// TwinCAT 3 PLC project PLC1
// ProgramVersion: 3.1.4024.0
// libraries:
//   Tc2_Standard, * (Beckhoff Automation GmbH)
//   Tc2_System, * (Beckhoff Automation GmbH)
//   Tc3_Module, * (Beckhoff Automation GmbH)
//   VisuDialogs, * (System)
//   VisuSymbols,3.5.10.0,System
// project tree:
//   / GlobalTextList.TcGTLO, PlcTask.TcTTO, Visualization Manager.TcVMO (not stored)
//   GVLs/ Cell.TcGVL, SEQ.TcGVL, VAL.TcGVL, Variables.TcGVL
//   POUs/ MAIN.TcPOU, POU.TcPOU, POU_1.TcPOU, FBAdd.TcPOU, Func.TcPOU, POU_3.TcPOU, SequencyControl.TcPOU, Simulation.TcPOU, ValveControl.TcPOU, Water_Tank.TcPOU
//   VISUs/ Header.TcVIS, MainScreen.TcVIS, Nav.TcVIS, Visualization.TcVIS, Visualization_1.TcVIS
// real-time tasks:
//   TASK PlcTask: cycle T#10ms, priority 20, ADS port 350
//   TASK VISU_TASK: cycle T#200000us, priority 30, ADS port 351

CONFIGURATION PLC1
    RESOURCE PLC ON TwinCAT3
        TASK PlcTask(INTERVAL := T#10ms, PRIORITY := 20);
        PROGRAM MAIN WITH PlcTask : MAIN;
    END_RESOURCE
END_CONFIGURATION

// ---- GVLs/Cell.TcGVL
{attribute 'qualified_only'}
VAR_GLOBAL
	bPalmButton:BOOL;
	bHousingPresent:BOOL;
	
END_VAR

// ---- GVLs/SEQ.TcGVL
{attribute 'qualified_only'}
VAR_GLOBAL
	iStepN:WORD;
	iSeqStepN: INT;
	sSeqStepDescription: STRING;
	bSeqStep_TaskDone: ARRAY[0..30] OF BOOL;
	fbSeqStepN_TaskDone_DelayTmr:ARRAY[0..30] OF TON;
	bSeqStepN_TaskDone_DelayDone:ARRAY[0..30] OF BOOL;

END_VAR

// ---- GVLs/VAL.TcGVL
{attribute 'qualified_only'}
VAR_GLOBAL
	bValve_A_WorkCmd:BOOL;
	bValve_A_HomeCmd:BOOL;
	bValve_A_AtWorkSensor:BOOL;
	bValve_A_AtHomeSensor:BOOL;
	
    bValve_B_WorkCmd:BOOL;
	bValve_B_HomeCmd:BOOL;
	bValve_B_AtWorkSensor:BOOL;
	bValve_B_AtHomeSensor:BOOL;
	
	bValve_C_WorkCmd:BOOL;
	bValve_C_HomeCmd:BOOL;
	bValve_C_AtWorkSensor:BOOL;
	bValve_C_AtHomeSensor:BOOL;
	
	bValve_D_WorkCmd:BOOL;
	bValve_D_HomeCmd:BOOL;
	bValve_D_AtWorkSensor:BOOL;
	bValve_D_AtHomeSensor:BOOL;
	
	bAllValves_At_Home:BOOL;
	
END_VAR

// ---- GVLs/Variables.TcGVL
{attribute 'qualified_only'}
VAR_GLOBAL
	stop:BOOL;
	start:BOOL;
	motor1:BOOL;
	motor2:BOOL;
	motor3:BOOL;
	LED:BOOL;
	Button:BOOL;
	Temp:BOOL;
END_VAR

// ---- POUs/MAIN.TcPOU
PROGRAM MAIN
VAR
END_VAR

SEQ.iStepN:=30;
Simulation();
POU();
Water_Tank();
POU_1();
POU_3();
SequencyControl();
ValveControl();

END_PROGRAM

// ---- POUs/Simulation.TcPOU
PROGRAM Simulation
VAR
END_VAR

VAL.bValve_A_AtHomeSensor:=VAL.bValve_A_HomeCmd;
VAL.bValve_A_AtWorkSensor:=VAL.bValve_A_WorkCmd;

VAL.bValve_B_AtHomeSensor:=VAL.bValve_B_HomeCmd;
VAL.bValve_B_AtWorkSensor:=VAL.bValve_B_WorkCmd;

VAL.bValve_C_AtHomeSensor:=VAL.bValve_C_HomeCmd;
VAL.bValve_C_AtWorkSensor:=VAL.bValve_C_WorkCmd;

VAL.bValve_D_AtHomeSensor:=VAL.bValve_D_HomeCmd;
VAL.bValve_D_AtWorkSensor:=VAL.bValve_D_WorkCmd;

END_PROGRAM

// ---- POUs/POU.TcPOU
PROGRAM POU
VAR
	T1: TON;
	TON_0:TON;
    Cycle: BOOL;
END_VAR
VAR // added by the converter: edge detectors and wires of the graphical bodies
    _w1 : BOOL;
END_VAR

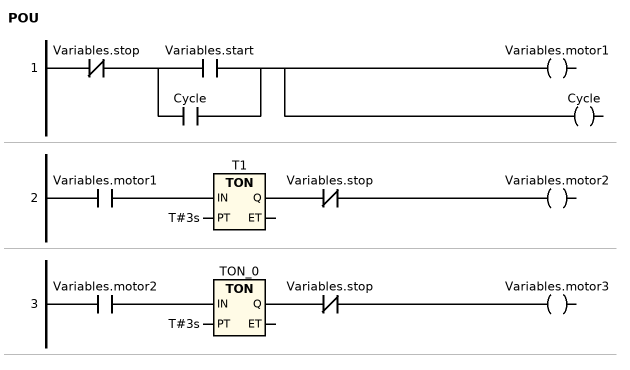
// NETWORK 1
_w1 := NOT Variables.stop AND (Variables.start OR Cycle);
Variables.motor1 := _w1;
Cycle := _w1;

// NETWORK 2
T1(IN := Variables.motor1, PT := T#3s); // TON
Variables.motor2 := T1.Q AND NOT Variables.stop;

// NETWORK 3
TON_0(IN := Variables.motor2, PT := T#3s); // TON
Variables.motor3 := TON_0.Q AND NOT Variables.stop;

END_PROGRAM

// ---- POUs/Water_Tank.TcPOU
PROGRAM Water_Tank
VAR
	start:BOOL;
	stop:BOOL;
	high:BOOL;
	low:BOOL;
	motor:BOOL;
	temp:BOOL;
	mix:BOOL;
	release:BOOL;
	
	TON_0: TON;
	TOF_0: TOF;
	TON_1: TON;
	MixFor10S: TOF;
	Delay2S: TON;
END_VAR

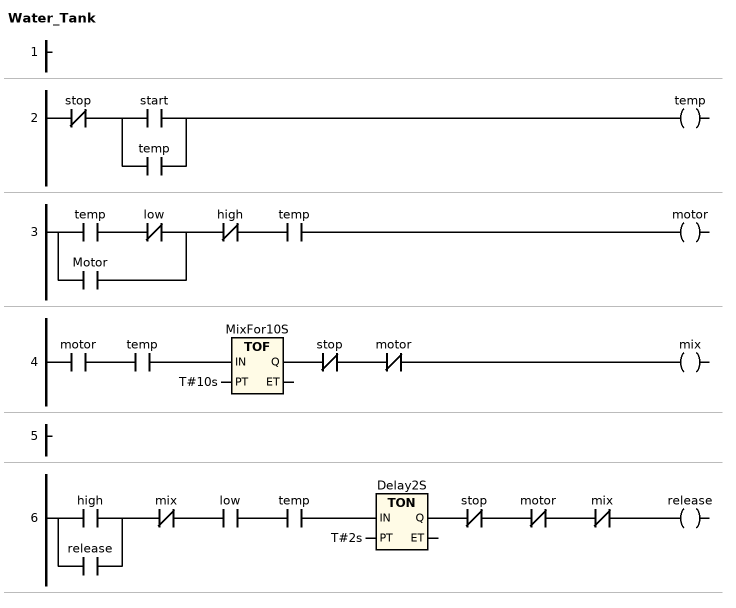
// NETWORK 1

// NETWORK 2
temp := NOT stop AND (start OR temp);

// NETWORK 3
motor := (temp AND NOT low OR Motor) AND NOT high AND temp;

// NETWORK 4
MixFor10S(IN := motor AND temp, PT := T#10s); // TOF
mix := MixFor10S.Q AND NOT stop AND NOT motor;

// NETWORK 5

// NETWORK 6
Delay2S(IN := (high OR release) AND NOT mix AND low AND temp, PT := T#2s); // TON
release := Delay2S.Q AND NOT stop AND NOT motor AND NOT mix;

END_PROGRAM

// ---- POUs/POU_1.TcPOU
PROGRAM POU_1
VAR
	x:BOOL;
	y:BOOL;
     rr:BOOL;
	 ss:bool;
	counter: CTU;
	coun:WORD;
END_VAR

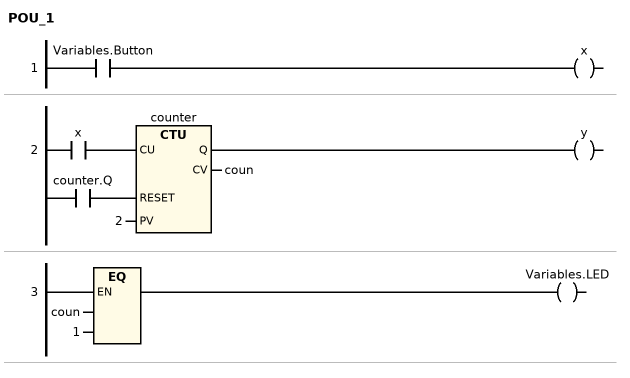
// NETWORK 1
x := Variables.Button;

// NETWORK 2
counter(CU := x, RESET := counter.Q, PV := 2, CV => coun); // CTU
y := counter.Q;

// NETWORK 3
Variables.LED := coun = 1;

END_PROGRAM

// ---- POUs/POU_3.TcPOU
PROGRAM POU_3
VAR
	count:WORD;
	prePushed:BOOL;
	pre: INT;
	fbCal:FBAdd;
	result:WORD;
	x:WORD;
	y:WORD;
	z:word;
END_VAR


IF Variables.Button THEN 
	IF NOT prePushed THEN
		count:=count+1;
		prePushed:=TRUE;
		Variables.LED:=NOT Variables.LED;
	END_IF
ELSE
	prePushed:=FALSE;	
END_IF
	
fbCal(a:=5,b:=3,c=>result);


x:=4;
y:=7;
//count:=Func(1,4);
z:=Func(x,y);

ACTION ACT:

END_ACTION

METHOD PUBLIC METH : BOOL
VAR_INPUT
END_VAR
END_METHOD

METHOD PUBLIC METH_1 : BOOL
VAR_INPUT
END_VAR
END_METHOD

END_PROGRAM

// ---- POUs/FBAdd.TcPOU
FUNCTION_BLOCK FINAL FBAdd
VAR_INPUT
	a:WORD;
	b:WORD;
END_VAR
VAR_OUTPUT
	c:word;
END_VAR
VAR
END_VAR

c:=a+b;
c:=a*b;

ACTION ACT:

END_ACTION

METHOD PUBLIC METH : BOOL
VAR_INPUT
END_VAR
END_METHOD

METHOD PRIVATE METH_1 : BOOL
VAR_INPUT
END_VAR
END_METHOD

PROPERTY PUBLIC Prop : INT
GET
END_GET
SET
END_SET
END_PROPERTY

END_FUNCTION_BLOCK

// ---- POUs/Func.TcPOU
FUNCTION Func : WORD
VAR_INPUT
	a:WORD;
	b:WORD;
END_VAR
VAR
	c:WORD;
END_VAR

c:=a+b;
Func:=c;
RETURN;

END_FUNCTION

// ---- POUs/SequencyControl.TcPOU
PROGRAM SequencyControl
VAR
	index:WORD;
END_VAR

CASE SEQ.iSeqStepN OF 
	 0:    //INIT
		 SEQ.sSeqStepDescription:='Init';
		 SEQ.bSeqStep_TaskDone[0]:=VAL.bAllValves_At_Home AND Cell.bHousingPresent AND Cell.bPalmButton;  //trigger the sequency
		 IF SEQ.bSeqStepN_TaskDone_DelayDone[0] THEN
			 FOR index:=1 TO SEQ.iStepN DO
				 SEQ.bSeqStep_TaskDone[index]:=FALSE;
			 END_FOR
			 seq.iSeqStepN:=5;
		 END_IF
	5:
		 SEQ.sSeqStepDescription:='Loading parts to hoursing';
		 SEQ.bSeqStep_TaskDone[5]:=VAL.bValve_A_AtWorkSensor;
		 IF SEQ.bSeqStepN_TaskDone_DelayDone[5] THEN
			 FOR index:=6 TO SEQ.iStepN DO
				 SEQ.bSeqStep_TaskDone[index]:=FALSE;
			 END_FOR
			 seq.iSeqStepN:=10;
		 END_IF
	10:
		 SEQ.sSeqStepDescription:='Clamp house';
		 SEQ.bSeqStep_TaskDone[10]:=VAL.bValve_A_AtWorkSensor AND VAl.bValve_B_AtWorkSensor;
		 IF SEQ.bSeqStepN_TaskDone_DelayDone[10] THEN
			 FOR index:=11 TO SEQ.iStepN DO
				 SEQ.bSeqStep_TaskDone[index]:=FALSE;
			 END_FOR
			 seq.iSeqStepN:=15;
		 END_IF
	15:
  	     SEQ.sSeqStepDescription:='Press/crimp the housing';
		 SEQ.bSeqStep_TaskDone[15]:=VAL.bValve_B_AtWorkSensor AND VAL.bValve_C_AtWorkSensor AND VAL.bValve_A_AtHomeSensor;
		 IF SEQ.bSeqStepN_TaskDone_DelayDone[15] THEN
			 FOR index:=0 TO SEQ.iStepN DO
				 SEQ.bSeqStep_TaskDone[index]:=FALSE;
			 END_FOR
			 seq.iSeqStepN:=20;
		 END_IF
	20:
  	     SEQ.sSeqStepDescription:='Open clamp';
		 SEQ.bSeqStep_TaskDone[20]:=VAl.bValve_B_AtHomeSensor;
		 IF SEQ.bSeqStepN_TaskDone_DelayDone[20] THEN
			 FOR index:=21 TO SEQ.iStepN DO
				 SEQ.bSeqStep_TaskDone[index]:=FALSE;
			 END_FOR
			 seq.iSeqStepN:=25;
		 END_IF
	25:  //work on cyl D
		 SEQ.sSeqStepDescription:='Heat houring for 10s';
		 SEQ.bSeqStep_TaskDone[25]:=VAL.bValve_D_AtWorkSensor AND VAL.bValve_C_AtWorkSensor;
		 IF SEQ.bSeqStepN_TaskDone_DelayDone[25] THEN
			 FOR index:=26 TO SEQ.iStepN DO
				 SEQ.bSeqStep_TaskDone[index]:=FALSE;
			 END_FOR
			 seq.iSeqStepN:=30;
		 END_IF
	30:  //home, home cyn C and Cyn B
		 SEQ.sSeqStepDescription:='Stop heat, open clamp';
		 SEQ.bSeqStep_TaskDone[30]:=VAL.bValve_C_AtHomeSensor AND VAL.bValve_D_AtHomeSensor;
		 IF SEQ.bSeqStepN_TaskDone_DelayDone[30] THEN
//			 FOR index:=26 TO SEQ.iStepN DO
//				 SEQ.bSeqStep_TaskDone[index]:=FALSE;
//			 END_FOR
			 seq.iSeqStepN:=0;
		 END_IF
END_CASE
SequencyCondition();

METHOD PUBLIC SequencyCondition : BOOL
VAR_INPUT
END_VAR
SEQ.fbSeqStepN_TaskDone_DelayTmr[0](IN:= SEQ.bSeqStep_TaskDone[0], PT:=T#2S , Q=>SEQ.bSeqStepN_TaskDone_DelayDone[0] );
SEQ.fbSeqStepN_TaskDone_DelayTmr[5](IN:= SEQ.bSeqStep_TaskDone[5], PT:=T#2S , Q=>SEQ.bSeqStepN_TaskDone_DelayDone[5] );
SEQ.fbSeqStepN_TaskDone_DelayTmr[10](IN:= SEQ.bSeqStep_TaskDone[10], PT:=T#2S , Q=>SEQ.bSeqStepN_TaskDone_DelayDone[10] );
SEQ.fbSeqStepN_TaskDone_DelayTmr[15](IN:= SEQ.bSeqStep_TaskDone[15], PT:=T#2S , Q=>SEQ.bSeqStepN_TaskDone_DelayDone[15] );
SEQ.fbSeqStepN_TaskDone_DelayTmr[20](IN:= SEQ.bSeqStep_TaskDone[20], PT:=T#2S , Q=>SEQ.bSeqStepN_TaskDone_DelayDone[20] );
SEQ.fbSeqStepN_TaskDone_DelayTmr[25](IN:= SEQ.bSeqStep_TaskDone[25], PT:=T#10S , Q=>SEQ.bSeqStepN_TaskDone_DelayDone[25] );
SEQ.fbSeqStepN_TaskDone_DelayTmr[30](IN:= SEQ.bSeqStep_TaskDone[30], PT:=T#2S , Q=>SEQ.bSeqStepN_TaskDone_DelayDone[30] );
END_METHOD

END_PROGRAM

// ---- POUs/ValveControl.TcPOU
PROGRAM ValveControl
VAR
END_VAR

IF (SEQ.iSeqStepN=0 OR SEQ.iSeqStepN=30) THEN
	VAL.bValve_A_HomeCmd:=TRUE;
	VAL.bValve_A_WorkCmd:=FALSE;
	VAL.bValve_B_HomeCmd:=TRUE;
	VAL.bValve_B_WorkCmd:=FALSE;
	VAL.bValve_C_HomeCmd:=TRUE;
	VAL.bValve_C_WorkCmd:=FALSE;
	VAL.bValve_D_HomeCmd:=TRUE;
	VAL.bValve_D_WorkCmd:=FALSE;
END_IF
//A
IF (SEQ.iSeqStepN=5 OR SEQ.iSeqStepN=10)THEN
	VAL.bValve_A_WorkCmd:=TRUE;
	VAL.bValve_A_HomeCmd :=FALSE;
ELSE
	VAL.bValve_A_WorkCmd:=FALSE;
	VAL.bValve_A_HomeCmd :=TRUE;
END_IF
//B
IF (SEQ.iSeqStepN=10 OR SEQ.iSeqStepN=15)THEN
	VAL.bValve_B_WorkCmd:=TRUE;
	VAL.bValve_B_HomeCmd :=FALSE;
ELSE
	VAL.bValve_B_WorkCmd:=FALSE;
	VAL.bValve_B_HomeCmd :=TRUE;	
END_IF
//C Valve
IF (SEQ.iSeqStepN>=15 AND SEQ.iSeqStepN<=25)THEN
	VAL.bValve_C_WorkCmd:=TRUE;
	VAL.bValve_C_HomeCmd :=FALSE;
ELSE
	VAL.bValve_C_WorkCmd:=FALSE;
	VAL.bValve_C_HomeCmd :=TRUE;	
END_IF

//D Valve
IF (SEQ.iSeqStepN=25)THEN
	VAL.bValve_D_WorkCmd:=TRUE;
	VAL.bValve_D_HomeCmd :=FALSE;
ELSE
	VAL.bValve_D_WorkCmd:=FALSE;
	VAL.bValve_D_HomeCmd :=TRUE;	
END_IF

////Home
//IF (SEQ.iSeqStepN=30)THEN
//	VAL.bValve_D_WorkCmd:=TRUE;
//	VAL.bValve_D_HomeCmd :=FALSE;
//ELSE
//	VAL.bValve_B_WorkCmd:=FALSE;
//	VAL.bValve_B_HomeCmd :=TRUE;	
VAL.bAllValves_At_Home:=VAL.bValve_A_AtHomeSensor AND VAL.bValve_B_AtHomeSensor AND VAL.bValve_C_AtHomeSensor AND VAL.bValve_D_AtHomeSensor;

END_PROGRAM

// ---- GlobalTextList.TcGTLO
TEXTLIST GlobalTextList
  863 = 'START'
END_TEXTLIST

// ---- VISUs/Header.TcVIS
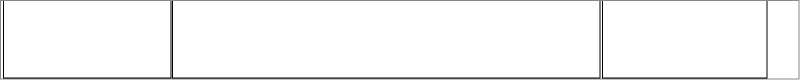
VISUALIZATION Header  // 800x80
    Rectangle (3,0 168x78)
    Rectangle (172,0 428x78)
    Rectangle (602,0 165x78)
END_VISUALIZATION

// ---- VISUs/MainScreen.TcVIS
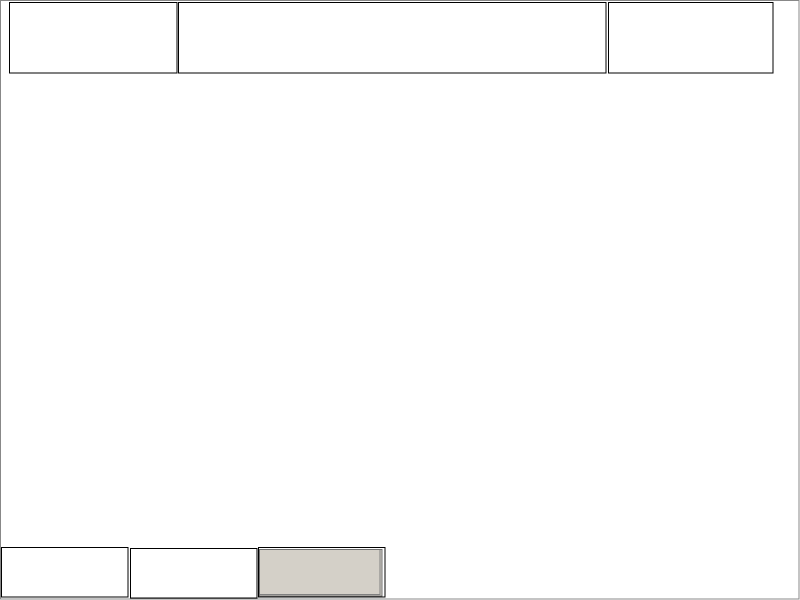
VISUALIZATION MainScreen  // 800x600
    Frame (6,2 800x73)
        shows Header()
    Frame (16,547 800x50)
        shows Nav()
END_VISUALIZATION

// ---- VISUs/Nav.TcVIS
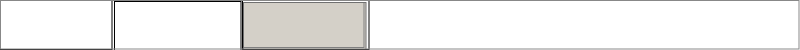
VISUALIZATION Nav  // 800x50
    Rectangle (-15,0 127x50)
    Rectangle (114,1 127x50)
    Rectangle (242,0 127x50)
    Button (243,2 123x47)
        OnMouseDown: change screen: Visualization
END_VISUALIZATION

// ---- VISUs/Visualization.TcVIS
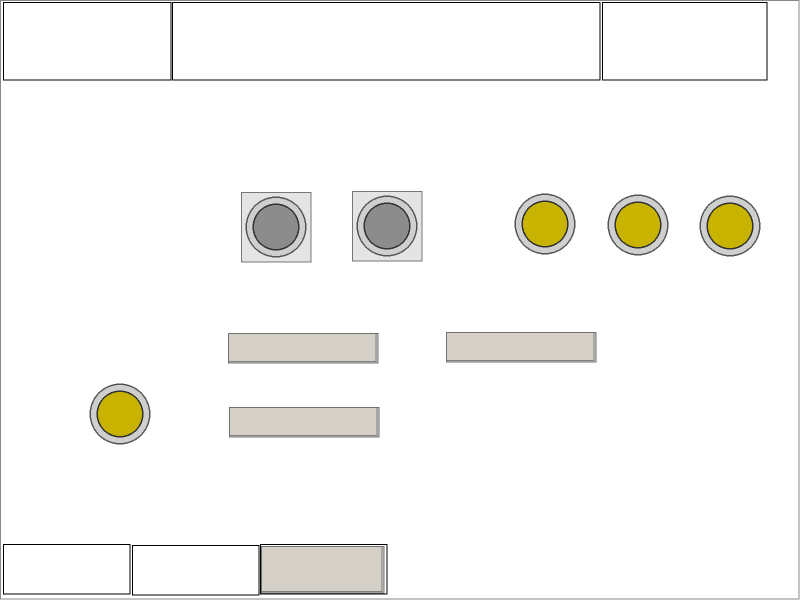
VISUALIZATION Visualization  // 800x600
    PushSwitch (241,192 70x70), variable: Variables.start, behaviour: TOGGLE, style: Switch-PushSwitch-Gray
    PushSwitch (352,191 70x70), variable: Variables.stop, behaviour: TOGGLE, style: Switch-PushSwitch-Gray
    Lamp1 (603,190 70x70), variable: Variables.motor2, style: Lamp-Lamp1-Yellow
    Lamp1 (510,189 70x70), variable: Variables.motor1, style: Lamp-Lamp1-Yellow
    Button (228,333 150x30)
        OnMouseDown: toggle Variables.start
        OnMouseUp: toggle Variables.start
    Lamp1 (695,191 70x70), variable: Variables.motor3, style: Lamp-Lamp1-Yellow
    Button (446,332 150x30)
        OnMouseDown: toggle Variables.stop
        OnMouseUp: toggle Variables.stop
    Lamp1 (85,379 70x70), variable: Variables.LED, style: Lamp-Lamp1-Yellow
    Button (229,407 150x30)
        OnMouseDown: toggle Variables.Button
        OnMouseUp: toggle Variables.Button
    Frame (0,2 800x80)
        shows Header()
    Frame (18,544 800x50)
        shows Nav()
END_VISUALIZATION

// ---- VISUs/Visualization_1.TcVIS
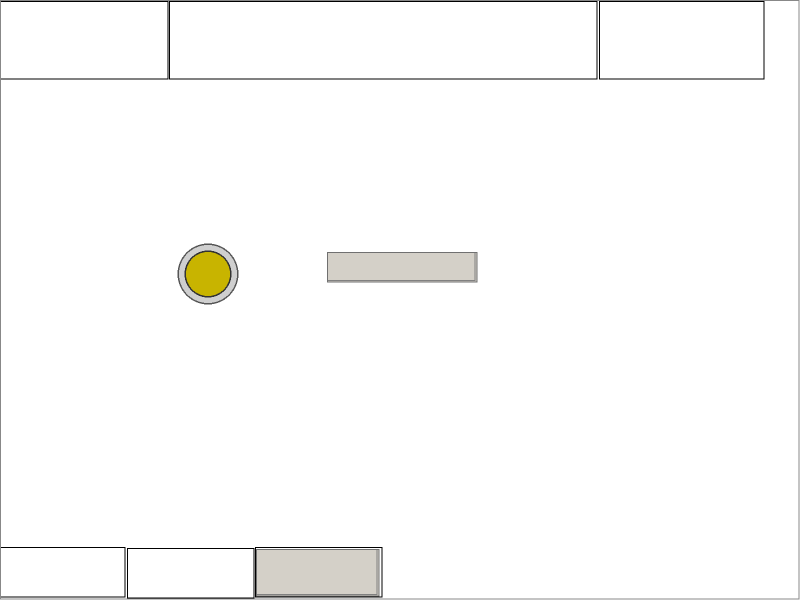
VISUALIZATION Visualization_1  // 800x600
    Button (327,252 150x30)
        OnMouseDown: toggle Variables.Button
        OnMouseUp: toggle Variables.Button
    Lamp1 (173,239 70x70), variable: Variables.LED, style: Lamp-Lamp1-Yellow
    Frame (-3,1 800x80)
        shows Header()
    Frame (13,547 800x50)
        shows Nav()
END_VISUALIZATION
